FUNCTION PushRegister : BOOL
VAR_INPUT
	arr : POINTER TO BYTE;
	numEntries : UDINT;
	entrySize : UDINT;
	
	newEntry : POINTER TO BYTE;
END_VAR
VAR_OUTPUT
	newIndex : UDINT;
END_VAR
VAR
	i : UDINT;
	
	arrSize : UDINT;
	
	test : BOOL;
END_VAR

arrSize := numEntries * entrySize;

FOR i:=0 TO arrSize-1 BY entrySize DO
	test := DataIsEmpty(arr:= ADR(arr[i]), arrSize:= entrySize);
	IF DataIsEmpty(arr:= ADR(arr[i]), arrSize:= entrySize) THEN
		test := MEMCPY(ADR(arr[i]), newEntry, entrySize) > 0;
		newIndex := i;
		PushRegister := TRUE;
	END_IF
		
END_FOR

END_FUNCTION

(* stored: Version 1.1.0.1, ProductVersion 3.1.4024.11
   POU PushRegister: Id {300492bd-f356-4b18-b166-bec49de8afde}, SpecialFunc None *)
